FUNCTION_BLOCK T_MockRoboConnect IMPLEMENTS I_RoboConnect
VAR_INPUT
  _error, _isBusy, _isDone, _isEnabled : BOOL;
  _errorId : UINT;
  _axisCount : UINT;
  _position, _toolPosition : ST_CartesianPoint;
END_VAR
VAR
  state, prevState : (INIT,
    IDLE,
    READY,
    ERROR_STATE) := INIT;

  initalised : BOOL;
  connectionTimer : TON;
  tasktimer : TON;
  _connection : I_Connection;
  _commandQueue : I_CommandQueue;
  _commandTask : T_MockCommandTask;
  _boolCommandTask : T_MockBoolCommandTask;
  _numberCommandTask : T_MockNumberCommandTask;

  digitalOutputs : ARRAY[1..DIGITAL_OUTPUT_COUNT] OF BOOL;
  digitalIntputs : ARRAY[1..DIGITAL_INPUT_COUNT] OF BOOL;
  analogOutputs : ARRAY[1..ANALOG_OUTPUT_COUNT] OF LREAL;
  analogIntputs : ARRAY[1..ANALOG_INPUT_COUNT] OF LREAL;

  toolDigitalOutputs : ARRAY[1..TOOL_DIGITAL_OUTPUT] OF BOOL;
  toolDigitalIntputs : ARRAY[1..TOOL_DIGITAL_INPUT] OF BOOL;
  toolAnalogOutputs : ARRAY[1..TOOL_ANALOG_INPUT] OF LREAL;
  toolAnalogIntputs : ARRAY[1..TOOL_ANALOG_OUTPUT] OF LREAL;

  axes : ARRAY[1..AXIS_COUNT] OF LREAL;

END_VAR
VAR CONSTANT
  DIGITAL_OUTPUT_COUNT : UINT := 6;
  DIGITAL_INPUT_COUNT : UINT := 6;
  ANALOG_INPUT_COUNT : UINT := 6;
  ANALOG_OUTPUT_COUNT : UINT := 6;
  TOOL_ANALOG_OUTPUT : UINT := 2;
  TOOL_DIGITAL_OUTPUT : UINT := 2;
  TOOL_ANALOG_INPUT : UINT := 2;
  TOOL_DIGITAL_INPUT : UINT := 2;
  AXIS_COUNT : UINT := 6;

END_VAR

PROPERTY Busy : BOOL
GET
END_GET
END_PROPERTY

PROPERTY CartesianPosition : TcRobot.ST_CartesianPoint
GET
END_GET
END_PROPERTY

METHOD ClearError : BOOL
VAR_OUTPUT
	task	: TcRobot.I_Task;
END_VAR
END_METHOD

METHOD Connect : BOOL
connectionTimer( IN := FALSE );
connectionTimer( IN := TRUE );
END_METHOD

PROPERTY Connected : BOOL
GET
Connected := connectionTimer.Q;
END_GET
END_PROPERTY

METHOD CyclicLogic
connectionTimer();
taskTimer();

IF taskTimer.Q THEN
  _commandTask(_Timeout := TRUE);
END_IF
END_METHOD

METHOD Disable : BOOL
VAR_OUTPUT
  task : I_Task;
END_VAR
VAR
  resultTask : T_CommandTask;
END_VAR
IF NOT connectionTimer.Q THEN
  task := resultTask;
  RETURN;
END_IF
END_METHOD

METHOD Disconnect : BOOL
VAR_OUTPUT
  task : I_Task;
END_VAR
connectionTimer( IN := FALSE );
END_METHOD

PROPERTY Done : BOOL
GET
END_GET
END_PROPERTY

METHOD Enable : BOOL
VAR_OUTPUT
  task : I_Task;
END_VAR
END_METHOD

PROPERTY Enabled : BOOL
GET
END_GET
END_PROPERTY

PROPERTY Error : BOOL
GET
END_GET
END_PROPERTY

PROPERTY ErrorID : LREAL
GET
END_GET
END_PROPERTY

METHOD GetAnalogOutput : BOOL
VAR_INPUT
  Index : UINT;
END_VAR
VAR_OUTPUT
  task : I_NumberResultTask;
END_VAR
IF Index < 1 OR index > ANALOG_OUTPUT_COUNT THEN
  GetAnalogOutput := FALSE;
  RETURN;
END_IF

_commandTask(_Result := analogOutputs[Index]);
task := _numberCommandTask;

GetAnalogOutput := TRUE;
END_METHOD

METHOD GetAxisCurrents : BOOL
VAR_IN_OUT
  Values : ARRAY[*] OF LREAL;
END_VAR
VAR_OUTPUT
  task : I_Task;
END_VAR
END_METHOD

METHOD GetAxisPositions : BOOL
VAR_IN_OUT
  Values : ARRAY[*] OF LREAL;
END_VAR
VAR_OUTPUT
  task : I_Task;
END_VAR
END_METHOD

METHOD GetAxisTemperatures : BOOL
VAR_IN_OUT
  Values : ARRAY[*] OF LREAL;
END_VAR
VAR_OUTPUT
  task : I_Task;
END_VAR
END_METHOD

METHOD GetDigitalOutput : BOOL
VAR_INPUT
    Index : UINT;
END_VAR
VAR_OUTPUT
  task : I_BoolResultTask;
  value : BOOL;
END_VAR
VAR
  cmdTask : T_CommandTask;
END_VAR
IF Index < 1 OR index > DIGITAL_OUTPUT_COUNT THEN
  GetDigitalOutput := FALSE;
  RETURN;
END_IF

_commandTask(_Result := TO_LREAL(digitalOutputs[Index]), _Done := TRUE);
task := _boolCommandTask;

GetDigitalOutput := TRUE;
END_METHOD

METHOD GetJointPositions : BOOL (* false if incompatible array length*)
VAR_IN_OUT
	(* values overwritten with joint positions.*)
	  joints : ARRAY[*] OF LREAL;
END_VAR
END_METHOD

METHOD GetToolAnalogOutput : BOOL
VAR_INPUT
    Index : UINT;
END_VAR
VAR_OUTPUT
  task : I_NumberResultTask;
END_VAR
IF Index < 1 OR index > DIGITAL_OUTPUT_COUNT THEN
  GetToolAnalogOutput := FALSE;
  RETURN;
END_IF

_commandTask(_Result := toolAnalogOutputs[Index]);
task := _numberCommandTask;

GetToolAnalogOutput := TRUE;
END_METHOD

METHOD GetToolDigitalOutput : BOOL
VAR_INPUT
	Index	: UINT;
END_VAR
VAR_OUTPUT
	task	: I_BoolResultTask;
END_VAR
IF Index < 1 OR Index > TOOL_DIGITAL_OUTPUT THEN
  GetToolDigitalOutput := FALSE;
  RETURN;
END_IF

_commandTask(_Result := TO_LREAL(toolDigitalOutputs[Index]));
task := _boolCommandTask;

GetToolDigitalOutput := TRUE;
END_METHOD

METHOD Halt : BOOL
VAR_OUTPUT
  task : I_Task;
END_VAR
END_METHOD

METHOD IsAtCartesianPosition : BOOL
VAR_INPUT
	point	: TcRobot.ST_CartesianPoint;
END_VAR
END_METHOD

METHOD IsAtJointPosition : BOOL
VAR_IN_OUT
	(* positions 1..NumberOfAxes will be used. passed array should be dimensioned accordingly*)
  joints : ARRAY[*] OF LREAL; // positions 1..NumberOfAxes will be used. passed array should be dimensioned accordingly
END_VAR
END_METHOD

METHOD JogAxis : BOOL // default tool and user frame
VAR_INPUT
  axisIndex : UDINT; // joint or enumerated cartesian direction/vector. See concrete type docs for enumeration of cartesian coords.
  axisDirection : BOOL; // TRUE = positive, FALSE = negative
  jogType : E_JogType; // Cartesian or Joint space
END_VAR
VAR_OUTPUT
	task	: TcRobot.I_Task;
END_VAR
END_METHOD

METHOD JogAxisAdvanced : BOOL
VAR_INPUT
  axisIndex : UDINT; // joint or enumerated cartesian direction/vector. See concrete type docs for enumeration of cartesian coords.
  axisDirection : BOOL; // TRUE = positive, FALSE = negative
  jogType : E_JogType; // Cartesian or Joint space
  coordType : INT; // set to 0 to leave default
  user : INT; // set to 0 to leave default
  tool : INT; // set to 0 to leave default
END_VAR
VAR_OUTPUT
	task	: TcRobot.I_Task;
END_VAR
END_METHOD

PROPERTY Manufacturer : STRING
GET
END_GET
END_PROPERTY

PROPERTY Model : STRING
GET
END_GET
END_PROPERTY

METHOD MoveAbs : BOOL
VAR_INPUT
  point : ST_CartesianPoint;
END_VAR
VAR_OUTPUT
  task : I_Task;
END_VAR
END_METHOD

METHOD MoveJ : BOOL
VAR_IN_OUT
  joints : ARRAY[*] OF LREAL;
END_VAR
VAR_OUTPUT
  task : I_Task;
END_VAR
VAR
  returnedTask : T_CommandTask;
END_VAR
IF UPPER_BOUND(joints,1) > _axisCount THEN
  task := returnedTask;
  RETURN;
END_IF
END_METHOD

PROPERTY Position : ST_CartesianPoint
GET
END_GET
END_PROPERTY

METHOD Reset : BOOL
VAR_OUTPUT
  task : I_Task;
END_VAR
END_METHOD

PROPERTY Running : BOOL
GET
END_GET
END_PROPERTY

METHOD SetAnalogOutput : BOOL
VAR_INPUT
  Index : UINT;
  Value : LREAL;
END_VAR
VAR_OUTPUT
  task : I_Task;
END_VAR
IF Index < 1 OR index > DIGITAL_OUTPUT_COUNT THEN
  SetAnalogOutput := FALSE;
  RETURN;
END_IF

tasktimer.IN := FALSE;
tasktimer.IN := TRUE;

analogOutputs[Index] := Value;
task := _commandTask;

SetAnalogOutput := TRUE;
END_METHOD

METHOD SetAtPosDeltas : BOOL
VAR_INPUT
  atPosCartesianDeltas : ST_CartesianPoint;
END_VAR
VAR_IN_OUT
  atPosJointDeltas : ARRAY[*] OF LREAL; // positions 1..NumberOfAxes will be used. passed array should be dimensioned accordingly
END_VAR
END_METHOD

METHOD SetBufferMode : BOOL
VAR_INPUT
  BufferMode : E_BufferMode;
END_VAR
END_METHOD

METHOD SetCarteasianAcceleration : BOOL
VAR_INPUT
  Acceleration : LREAL;
END_VAR
VAR_OUTPUT
  task : I_Task;
END_VAR
END_METHOD

METHOD SetCartesianSpeed : BOOL
VAR_INPUT
  Speed : LREAL;
END_VAR
VAR_OUTPUT
  task : I_Task;
END_VAR
END_METHOD

METHOD PUBLIC SetConnectionTime  // set simulated connection time
VAR_INPUT
  connectionTime : TIME;
END_VAR
connectionTimer.PT := connectionTime;
END_METHOD

METHOD SetDigitalOutput : BOOL
VAR_INPUT
  Index : UINT;
  Value : BOOL;
END_VAR
VAR_OUTPUT
  task : I_Task;
END_VAR
IF Index < 1 OR index > DIGITAL_OUTPUT_COUNT THEN
  SetDigitalOutput := FALSE;
  RETURN;
END_IF

tasktimer.IN := FALSE;
tasktimer.IN := TRUE;

digitalOutputs[Index] := TRUE;
_commandTask(_Done := TRUE);
task := _commandTask;

SetDigitalOutput := TRUE;
END_METHOD

METHOD PUBLIC SetGeneralCommandResponseDuration : BOOL // This sets the duration that the task will take, used for causing timeout or done in the returned task
VAR_INPUT
    taskTime : TIME;
END_VAR
tasktimer.PT := taskTime;
END_METHOD

METHOD SetJogType : BOOL
VAR_INPUT
  JogType : E_JogType;
END_VAR
VAR_OUTPUT
  task : I_Task;
END_VAR
END_METHOD

METHOD SetJointAcceleration : BOOL
VAR_INPUT
  Acceleration : LREAL;
END_VAR
VAR_OUTPUT
  task : I_Task;
END_VAR
END_METHOD

METHOD SetJointSpeed : BOOL
VAR_INPUT
  Speed : LREAL;
END_VAR
VAR_OUTPUT
  task : I_Task;
END_VAR
END_METHOD

METHOD SetToolAnalogOutput : BOOL
VAR_INPUT
  Index : UINT;
  Value : LREAL;
END_VAR
VAR_OUTPUT
  task : I_Task;
END_VAR
IF Index > ANALOG_OUTPUT_COUNT THEN
  SetToolAnalogOutput := FALSE;
  RETURN;
END_IF

tasktimer.IN := FALSE;
tasktimer.IN := TRUE;

toolDigitalOutputs[Index] := TRUE;
task := _commandTask;

SetToolAnalogOutput := TRUE;
END_METHOD

METHOD SetToolDigitalOutput : BOOL
VAR_INPUT
	Index	: UINT;
	Value	: BOOL;
END_VAR
VAR_OUTPUT
	task	: TcRobot.I_Task;
END_VAR
IF Index < 1 OR Index > TOOL_ANALOG_OUTPUT THEN
  SetToolDigitalOutput := FALSE;
  RETURN;
END_IF

tasktimer.IN := FALSE;
tasktimer.IN := TRUE;

toolDigitalOutputs[Index] := TRUE;
task := _commandTask;

SetToolDigitalOutput := TRUE;
END_METHOD

METHOD SetToolFrame : BOOL
VAR_INPUT
 Frame : ST_CartesianPoint;
END_VAR
VAR_OUTPUT
  task : I_Task;
END_VAR
END_METHOD

METHOD SetTransitionMode : BOOL
VAR_INPUT
END_VAR
END_METHOD

METHOD SetTransitionParameter : BOOL
VAR_INPUT
  CPratio : LREAL;
END_VAR
VAR_OUTPUT
	task	: TcRobot.I_Task;
END_VAR
END_METHOD

METHOD SetUserFrame : BOOL
VAR_INPUT
  Frame : ST_CartesianPoint;
END_VAR
VAR_OUTPUT
	task : I_Task;
END_VAR
END_METHOD

METHOD Stop : BOOL
VAR_OUTPUT
  task : I_Task;
END_VAR
END_METHOD

PROPERTY ToolPosition : ST_CartesianPoint
GET
END_GET
END_PROPERTY

END_FUNCTION_BLOCK

(* stored: Version 1.1.0.1
   POU T_MockTcRobot: Id {201056d0-98c2-4ff9-b470-1c80ccf83dde}, SpecialFunc None
   Folder Methods: Id {633a559d-0be4-494e-b564-dfbde4c320fd}
   Folder MockSetup Methods: Id {6663e216-8a27-0428-0e05-3423509a4f3d}
   Folder Properties: Id {439c51c2-74ab-420d-a2ce-c5c3c04fd93e}
   Property Busy: Id {be087c2b-05e3-4b2b-9cd2-e6c0fd449973}
   Get Get: Id {f9b28191-c884-4748-ad02-67f19cd6df5e}
   Property CartesianPosition: Id {7ad9454c-f24d-41c7-a977-f0d5ba108681}
   Get Get: Id {3cabd2f2-3f58-42e5-81b1-95d14c25f156}
   Method ClearError: Id {8a001a36-ca9f-4d28-b7f6-458e76a98629}
   Method Connect: Id {52902f6d-f80f-48b4-9f6a-82181fc37f94}
   Property Connected: Id {ee21ccfd-ba7b-4f6a-bed3-758d5b62f035}
   Get Get: Id {4c45a3ef-8fb0-4369-9427-31f87248cd96}
   Method CyclicLogic: Id {c3fd3be3-ccd9-4e33-b12c-93d2902836d6}
   Method Disable: Id {4cfdcbd7-25fa-486d-85c1-d89c75300fb4}
   Method Disconnect: Id {8ecd6e57-49e1-43b3-9652-a1b288dd9406}
   Property Done: Id {7d88ea25-3f3a-4514-9ad2-cae4e11952a8}
   Get Get: Id {69a1b751-1458-4825-91cc-b9dcc818c159}
   Method Enable: Id {34b8f714-1bc9-4d3d-a330-ff89ad98408e}
   Property Enabled: Id {fc0fc101-25a6-454b-bdc3-3f7e326f2a26}
   Get Get: Id {1ba6c64f-b764-4ed1-9ce3-08a066388529}
   Property Error: Id {c9dc4358-c962-4b68-bb6b-6600ddb8f5df}
   Get Get: Id {7f2055a5-d2dc-4571-a026-3c146bb3f237}
   Property ErrorID: Id {08d3ebdb-b083-44b2-87cf-732b45b21f29}
   Get Get: Id {521b1f8d-0d82-4ec1-b756-f45933e08951}
   Method GetAnalogOutput: Id {b322adc4-b30c-475c-bdb0-2ba7c39039ff}
   Method GetAxisCurrents: Id {fc570068-f9db-4768-89b4-60478ec9c0bd}
   Method GetAxisPositions: Id {9c14ea6f-f971-4dc2-8221-4e4e2b31db47}
   Method GetAxisTemperatures: Id {a731a00e-3c0a-4add-a96e-fd6d088806a4}
   Method GetDigitalOutput: Id {ddbb5b8f-52c5-4a9e-9e34-c18db80e0bb7}
   Method GetJointPositions: Id {2b8e9a86-fd78-4344-bbcd-0fe200aeddff}
   Method GetToolAnalogOutput: Id {a38a8162-0215-4ad4-8431-0a01d847acab}
   Method GetToolDigitalOutput: Id {9fffe7f0-c2a7-4f4c-b409-0dc3cc98c25a}
   Method Halt: Id {1f522c86-80d1-4428-8c2f-7a8c2666651f}
   Method IsAtCartesianPosition: Id {59686771-36ce-477f-a2c6-1bfff4544c83}
   Method IsAtJointPosition: Id {66eeedb0-7209-45b2-a6b3-aef2e7cfc684}
   Method JogAxis: Id {b723cea3-a58a-4642-b130-fa322bd8cf68}
   Method JogAxisAdvanced: Id {e76e1b11-ff2c-435b-add1-b9ad4ad224b9}
   Property Manufacturer: Id {5a43e0e0-9e77-485f-87c5-6338e32ed17c}
   Get Get: Id {482f138d-a761-4bc4-9125-978d3d017e01}
   Property Model: Id {f435e915-f498-42ff-80e0-2fc6bbbd32d6}
   Get Get: Id {26e6127e-5430-4f7c-aa44-95b7846ec867}
   Method MoveAbs: Id {d11a239e-0a9a-448a-9962-1a53a98ca5c5}
   Method MoveJ: Id {e423add9-81f9-4a51-b009-a07e53ce789c}
   Property Position: Id {46e2c8c4-9558-4310-a2a6-01359d992138}
   Get Get: Id {2173d570-f97d-4a42-8860-7c15f029019e}
   Method Reset: Id {421d94c9-1118-40da-8183-faff553dace0}
   Property Running: Id {0dacab0c-ea40-4e36-9cb5-0ef3bcd26dc6}
   Get Get: Id {d1d03029-a131-48f5-8644-b7baf860776a}
   Method SetAnalogOutput: Id {f79fae92-208b-48bb-a70b-40fc0ffe9ad6}
   Method SetAtPosDeltas: Id {c0f75a41-7ffc-4039-a90b-ce89194695b4}
   Method SetBufferMode: Id {6ffd794f-d6a9-4eb4-b470-6b664c06957e}
   Method SetCarteasianAcceleration: Id {85dda38a-040b-4f52-9ac5-51cddf3a9b78}
   Method SetCartesianSpeed: Id {fe07bbab-44d4-4192-af0e-5610faa953a3}
   Method SetConnectionTime: Id {33f430ae-2a96-0805-2f4e-abac8935e778}
   Method SetDigitalOutput: Id {fbad9e30-660d-44ee-b1e4-f426c3bf60ed}
   Method SetGeneralCommandResponseDuration: Id {8118186d-6855-4c8a-b59c-b7b713f02e50}
   Method SetJogType: Id {e28db961-d258-4313-8a33-3c20de35ebc8}
   Method SetJointAcceleration: Id {e49ec01e-e14d-437c-a820-aaa73f0c038c}
   Method SetJointSpeed: Id {b2f3ce57-58aa-4357-b698-11e54a0f9ec8}
   Method SetToolAnalogOutput: Id {39b00a63-134a-43a3-b689-a049deccd970}
   Method SetToolDigitalOutput: Id {a799ef3c-8388-4a9a-bef2-22e024f79347}
   Method SetToolFrame: Id {7845f72d-20ab-41f5-a329-3c9bfd0fd8fb}
   Method SetTransitionMode: Id {39572f02-5f91-423e-a853-b22d710b61f5}
   Method SetTransitionParameter: Id {8775b29d-f761-40b1-ac4f-383a3c43ae28}
   Method SetUserFrame: Id {b885c6dd-241e-4063-921e-c573396ee25f}
   Method Stop: Id {b6470bbe-62bc-49e9-8f0d-e53ffab7abb5}
   Property ToolPosition: Id {d4b202f9-68fe-4baf-a062-65718cfd8d98}
   Get Get: Id {69eba617-2635-4b58-851f-90f8212eff16} *)
